Fanuc KAREL source: ks00027.KL

-- PROVISIONAL review KL for V1013-1; original PC SHA256 fac1533f66cf746f2db85fa9db5ac435782a205a47d4e809d72117a031bdbdec
-- Incomplete behavior may be omitted. Consult companion uncertainty JSON. Do not deploy.
PROGRAM KS00027
%NOLOCKGROUP
VAR
  FLAG : BOOLEAN
  N : INTEGER
  STATUS : INTEGER
  PN : STRING[80]
  VN : STRING[80]
-- UNRESOLVED_DECL A type=001101
-- UNRESOLVED_DECL B type=001101
BEGIN
  -- UNRESOLVED_PC offsets 5-13; opcodes 3F,75
  -- UNRESOLVED_PC offsets 18-27; opcodes 3F,75
  -- UNRESOLVED_PC offsets 32-70; opcodes 27,22,22,2A,22,2A,22,22,AF
  -- UNRESOLVED_PC offsets 75-79; opcodes 7F
END KS00027
